FUNCTION_BLOCK CONVEYOR_DS_TS
  {SET_ATTRIBUTE(OpcUa, SERVICE)}
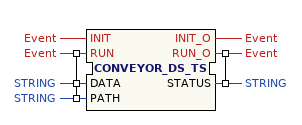
  EVENT_INPUT
    INIT;
    RUN WITH DATA, PATH; {SET_ATTRIBUTE(OpcUa, Method)}
  END_EVENT
  EVENT_OUTPUT
    INIT_O;
    RUN_O WITH STATUS;
  END_EVENT
  VAR_INPUT
    DATA : STRING;
    PATH : STRING;
  END_VAR
  VAR_OUTPUT
    STATUS : STRING;
  END_VAR
END_FUNCTION_BLOCK
